TYPE ST_DosingResults :
STRUCT
	iPump 		: USINT;
	iCheck		: USINT;
	rResult 	: LREAL;
	iRevs		: LREAL;
END_STRUCT
END_TYPE

(* stored: Version 1.1.0.1, ProductVersion 3.1.4024.15
   DUT ST_DosingResults: Id {de71ea9e-257d-47b6-8215-7717a7752470} *)
